Staubli VAL3: iGripClosed.pgx

public program iGripClosed(num& nNum[] (dimensions=1))
begin
  nNum=dioGet(iGripClosed)
end
